INTERFACE ITF_BaseCommand

END_INTERFACE

(* stored: Version 1.1.0.1
   Itf ITF_BaseCommand: Id {9d7c8a65-e020-0961-14d5-ad0889f068cf} *)
